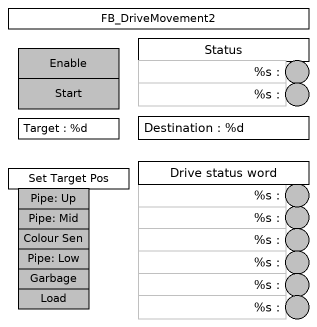
rectangle at (0,0)-(301,21): text "FB_DriveMovement2"
embedded screen at (130,30)-(301,311): FB_VC_Drive_Status
rectangle at (10,110)-(111,131): text "Target : %d"; shows $FB$.wTarget
rectangle at (10,40)-(111,71): text "Enable"; alarm colour if $FB$.bEnable; toggles $FB$.bEnable
rectangle at (10,70)-(111,101): text "Start"; alarm colour if $FB$.bStart; toggles $FB$.bStart
rectangle at (10,280)-(81,301): text "Load"; alarm colour if $FB$.wTarget = .GPOS_LOADING; runs INTERN ASSIGN $FB$.wTarget:=(GPOS_LOADING)
rectangle at (10,260)-(81,281): text "Garbage"; alarm colour if $FB$.wTarget = .GPOS_GARBAGE; runs INTERN ASSIGN $FB$.wTarget:=(GPOS_GARBAGE)
rectangle at (0,160)-(121,181): text "Set Target Pos"
rectangle at (10,240)-(81,261): text "Pipe: Low"; alarm colour if $FB$.wTarget = .GPOS_PIPE_LOW; runs INTERN ASSIGN $FB$.wTarget:=(GPOS_PIPE_LOW)
rectangle at (10,220)-(81,241): text "Colour Sen"; alarm colour if $FB$.wTarget = .GPOS_COLOR_SEN; runs INTERN ASSIGN $FB$.wTarget:=(GPOS_COLOR_SEN)
rectangle at (10,200)-(81,221): text "Pipe: Mid"; alarm colour if $FB$.wTarget = .GPOS_PIPE_MID; runs INTERN ASSIGN $FB$.wTarget:=(GPOS_PIPE_MID)
rectangle at (10,180)-(81,201): text "Pipe: Up"; alarm colour if $FB$.wTarget = .GPOS_PIPE_UP; runs INTERN ASSIGN $FB$.wTarget:=(GPOS_PIPE_UP)
1 more shapes without text or variables
*)

(* Visualisation FBs_Visu/FB_VC_Drive_Status
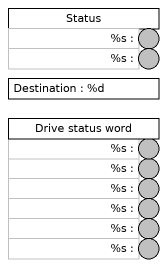
embedded screen at (0,150)-(151,171): VC_BOOLEANSTATUS
rectangle at (0,0)-(151,21): text "Status"
embedded screen at (0,170)-(151,191): VC_BOOLEANSTATUS
embedded screen at (0,130)-(151,151): VC_BOOLEANSTATUS
embedded screen at (0,190)-(151,211): VC_BOOLEANSTATUS
embedded screen at (0,210)-(151,231): VC_BOOLEANSTATUS
embedded screen at (0,230)-(151,251): VC_BOOLEANSTATUS
rectangle at (0,70)-(151,91): text "Destination : %d"; shows $FB$.wDestination
rectangle at (0,110)-(151,131): text "Drive status word"
embedded screen at (0,20)-(151,41): VC_BOOLEANSTATUS
embedded screen at (0,40)-(151,61): VC_BOOLEANSTATUS
*)

(* Visualisation Simulation/Simu_VC_Virtual_Ball
1 elements of other kinds (tables, trends, ...) not read
*)

(* Visualisation V_Drive
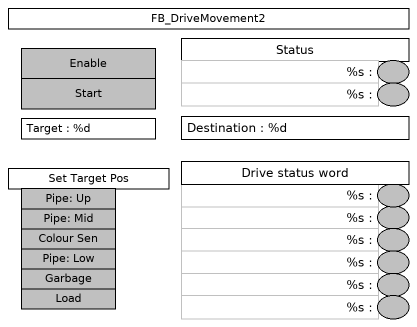
embedded screen at (0,0)-(401,311): FB_DriveMovement2
*)

(* Visualisation V_MAIN
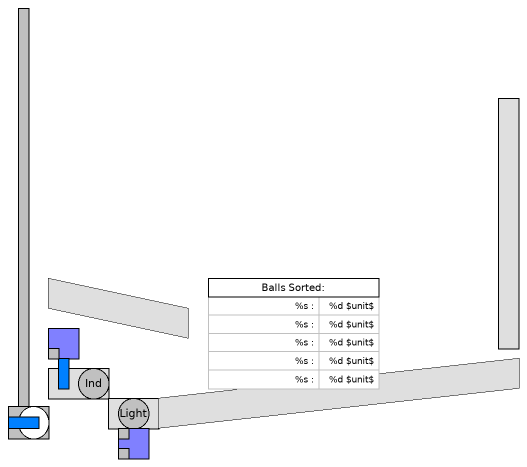
embedded screen at (60,320)-(531,451): VC_Graph_Sorter
embedded screen at (20,0)-(61,431): VC_Graph_Lift
embedded screen at (220,270)-(391,381): VC_Graph_Counters
2 more shapes without text or variables
*)

(* Visualisation V_VIRTUAL_MACHINE
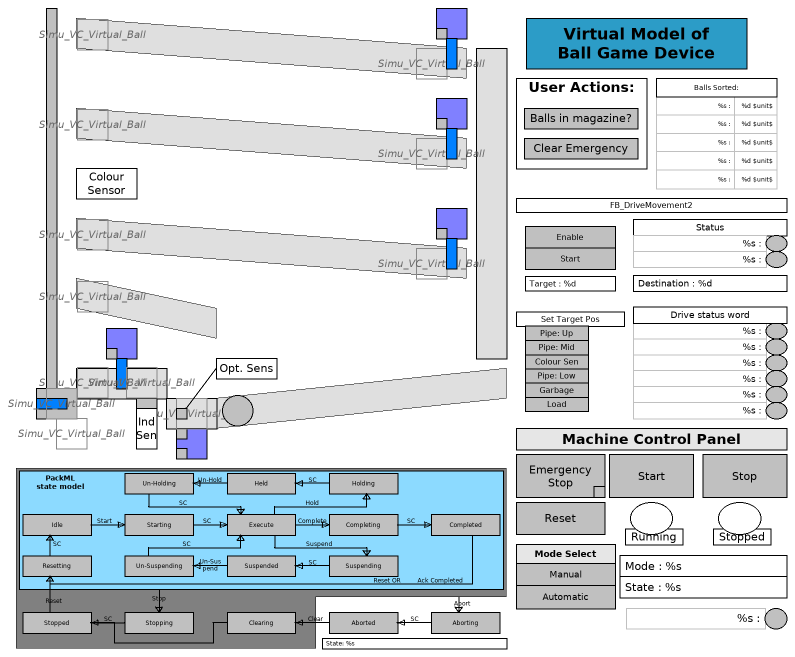
rectangle at (150,390)-(201,421): y offset -1 * PRG_HMI.iSorterLiftPos
rectangle at (100,350)-(111,381): invisible if .OSorterGate
rectangle at (120,390)-(141,401): alarm colour if .ISensorInd
rectangle at (160,420)-(171,431): alarm colour if .ISorterLiftUp
rectangle at (160,440)-(171,451): alarm colour if .ISorterLiftDown
rectangle at (90,340)-(101,351): alarm colour if .ISorterGateClosed
embedded screen at (160,390)-(191,421): Simu_VC_Virtual_Ball
rectangle at (160,400)-(171,411): alarm colour if .ISensorOpt
embedded screen at (110,359)-(141,390): Simu_VC_Virtual_Ball
embedded screen at (61,359)-(92,390): Simu_VC_Virtual_Ball
embedded screen at (40,410)-(71,441): Simu_VC_Virtual_Ball
rectangle at (20,380)-(61,411): y offset -1 * Simu_PRG_Simulation.iVirtualLiftPos
rectangle at (20,390)-(51,401): invisible if NOT .OEjector; y offset -1 * Simu_PRG_Simulation.iVirtualLiftPos
embedded screen at (30,380)-(61,411): Simu_VC_Virtual_Ball
embedded screen at (61,273)-(92,304): Simu_VC_Virtual_Ball
embedded screen at (61,211)-(92,242): Simu_VC_Virtual_Ball
embedded screen at (61,101)-(92,132): Simu_VC_Virtual_Ball
embedded screen at (61,11)-(92,42): Simu_VC_Virtual_Ball
embedded screen at (400,40)-(431,71): Simu_VC_Virtual_Ball
embedded screen at (400,130)-(431,161): Simu_VC_Virtual_Ball
embedded screen at (400,240)-(431,271): Simu_VC_Virtual_Ball
rectangle at (60,160)-(121,191): text "Colour / Sensor"
rectangle at (510,10)-(731,61): text "Virtual Model of / Ball Game Device"
rectangle at (120,400)-(141,441): text "Ind / Sen"
rectangle at (200,350)-(261,371): text "Opt. Sens"
ellipse at (206,387)-(237,418): invisible if NOT Simu_PRG_Simulation.bHasBallsInMagazine
embedded screen at (0,460)-(491,641): VC_PackMLStates
embedded screen at (640,70)-(761,181): VC_Graph_Counters
embedded screen at (500,190)-(771,411): FB_DriveMovement2
embedded screen at (500,420)-(771,601): VC_PANEL_MACHINECONTROL
rectangle at (420,220)-(431,231): alarm colour if .IGateClosedLow
rectangle at (420,110)-(431,121): alarm colour if .IGateClosedMid
rectangle at (420,20)-(431,31): alarm colour if .IGateClosedUp
rectangle at (430,120)-(441,151): invisible if .OGateMid
rectangle at (430,30)-(441,61): invisible if .OGateUp
rectangle at (430,230)-(441,261): invisible if .OGateLow
group at (500,70)-(631,161)
  rounded rectangle at (0,0)-(131,91): text "User Actions:"
  rounded rectangle at (8,30)-(122,51): text "Balls in magazine?"; alarm colour if Simu_PRG_Simulation.bHasBallsInMagazine; toggles Simu_PRG_Simulation.bHasBallsInMagazine
  rounded rectangle at (8,60)-(122,81): text "Clear Emergency"; alarm colour if NOT .IEmergencyClear; toggles .IEmergencyClear
embedded screen at (610,600)-(771,621): VC_BOOLEANSTATUS
19 more shapes without text or variables
*)

(* Visualisation Components/VC_BOOLEANSTATUS
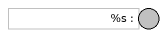
rectangle at (0,0)-(131,21): text "%s :"; shows $Name$
ellipse at (130,0)-(151,21): alarm colour if $bFlag$
*)

(* Visualisation Components/VC_Graph_Counters
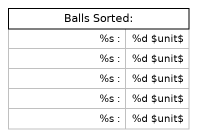
embedded screen at (0,20)-(181,41): VC_Var_Int
rectangle at (0,0)-(181,21): text "Balls Sorted:"
embedded screen at (0,40)-(181,61): VC_Var_Int
embedded screen at (0,60)-(181,81): VC_Var_Int
embedded screen at (0,80)-(181,101): VC_Var_Int
embedded screen at (0,100)-(181,121): VC_Var_Int
*)

(* Visualisation Components/VC_GRAPH_LIFT
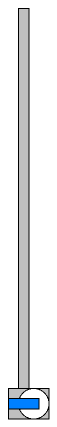
rectangle at (0,380)-(41,411): y offset -1 * PRG_HMI.iLiftPos
ellipse at (10,380)-(41,411): invisible if NOT .PRG_HMI.bBall_InLift; y offset -1 * PRG_HMI.iLiftPos
rectangle at (0,390)-(31,401): invisible if NOT .OEjector; y offset -1 * PRG_HMI.iLiftPos
1 more shapes without text or variables
*)

(* Visualisation Components/VC_GRAPH_SORTER
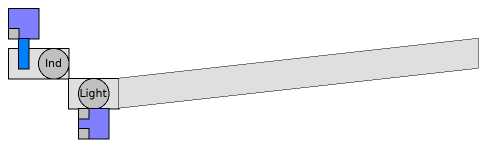
rectangle at (60,70)-(111,101): y offset -1 * PRG_HMI.iSorterLiftPos
rectangle at (10,30)-(21,61): invisible if .OSorterGate
ellipse at (70,70)-(101,101): text "Light"; alarm colour if .ISensorOpt; y offset -1 * PRG_HMI.iSorterLiftPos
ellipse at (30,40)-(61,71): text "Ind"; alarm colour if .ISensorInd
rectangle at (70,100)-(81,111): alarm colour if .ISorterLiftUp
rectangle at (70,120)-(81,131): alarm colour if .ISorterLiftDown
rectangle at (0,20)-(11,31): alarm colour if .ISorterGateClosed
6 more shapes without text or variables
*)

(* Visualisation Visual Components/VC_PackMLStates
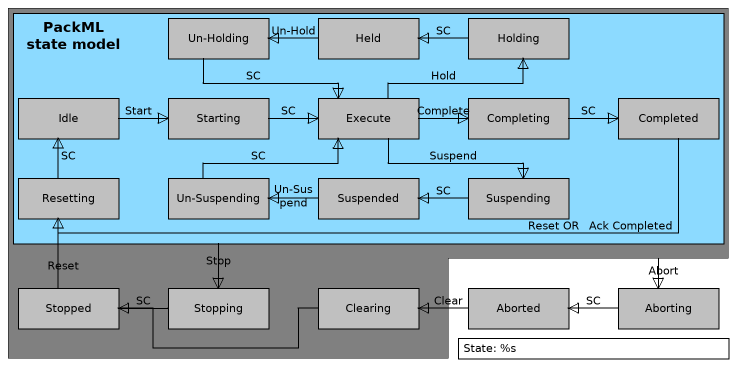
rounded rectangle at (160,280)-(261,321): text "Stopping"; alarm colour if $PackML$.eState = 4
rounded rectangle at (10,90)-(111,131): text "Idle"; alarm colour if $PackML$.eState = 6
rounded rectangle at (160,170)-(261,211): text "Un-Suspending"; alarm colour if $PackML$.eState = 11
rounded rectangle at (610,280)-(711,321): text "Aborting"; alarm colour if $PackML$.eState = 0
rounded rectangle at (460,280)-(561,321): text "Aborted"; alarm colour if $PackML$.eState = 1
rectangle at (450,330)-(721,351): text "State: %s"; shows .fbStateModel.eState
rounded rectangle at (310,280)-(411,321): text "Clearing"; alarm colour if $PackML$.eState = 2
rounded rectangle at (10,280)-(111,321): text "Stopped"; alarm colour if $PackML$.eState = 3
rounded rectangle at (10,170)-(111,211): text "Resetting"; alarm colour if $PackML$.eState = 5
rounded rectangle at (160,90)-(261,131): text "Starting"; alarm colour if $PackML$.eState = 7
rounded rectangle at (310,90)-(411,131): text "Execute"; alarm colour if $PackML$.eState = 8
rounded rectangle at (460,90)-(561,131): text "Completing"; alarm colour if $PackML$.eState = 15
rounded rectangle at (610,90)-(711,131): text "Completed"; alarm colour if $PackML$.eState = 16
rounded rectangle at (310,170)-(411,211): text "Suspended"; alarm colour if $PackML$.eState = 10
rounded rectangle at (460,170)-(561,211): text "Suspending"; alarm colour if $PackML$.eState = 9
rounded rectangle at (460,10)-(561,51): text "Holding"; alarm colour if $PackML$.eState = 12
rounded rectangle at (310,10)-(411,51): text "Held"; alarm colour if $PackML$.eState = 13
rounded rectangle at (160,10)-(261,51): text "Un-Holding"; alarm colour if $PackML$.eState = 14
polyline at (645,250)-(655,280): alarm colour if $PackML$.bAbort
rectangle at (635,255)-(676,271): text "Abort"; alarm colour if $PackML$.bAbort
polyline at (205,235)-(215,280): alarm colour if $PackML$.bStop
rectangle at (190,245)-(231,261): text "Stop"; alarm colour if $PackML$.bStop
polyline at (195,130)-(335,170): alarm colour if $PackML$.bSC
rectangle at (235,140)-(266,156): text "SC"; alarm colour if $PackML$.bSC
polyline at (195,50)-(335,90): alarm colour if $PackML$.bSC
polyline at (380,50)-(520,90): alarm colour if $PackML$.bHold
rectangle at (420,60)-(451,76): text "Hold"; alarm colour if $PackML$.bHold
polyline at (560,295)-(610,305): alarm colour if $PackML$.bSC
polyline at (45,210)-(55,280): alarm colour if $PackML$.bReset
polyline at (110,105)-(160,115): alarm colour if $PackML$.bStart
polyline at (110,295)-(310,340): alarm colour if $PackML$.bSC
rectangle at (230,60)-(261,76): text "SC"; alarm colour if $PackML$.bSC
polyline at (380,130)-(520,170): alarm colour if $PackML$.bSuspend
rectangle at (415,140)-(476,156): text "Suspend"; alarm colour if $PackML$.bSuspend
rectangle at (120,285)-(151,301): text "SC"; alarm colour if $PackML$.bSC
rectangle at (570,285)-(601,301): text "SC"; alarm colour if $PackML$.bSC
polyline at (410,295)-(460,305): alarm colour if $PackML$.bClear
rectangle at (420,285)-(461,301): text "Clear"; alarm colour if $PackML$.bClear
polyline at (260,105)-(310,115): alarm colour if $PackML$.bSC
rectangle at (265,95)-(296,111): text "SC"; alarm colour if $PackML$.bSC
rectangle at (110,95)-(151,111): text "Start"; alarm colour if $PackML$.bStart
rectangle at (35,250)-(76,266): text "Reset"; alarm colour if $PackML$.bReset
polyline at (410,185)-(460,195): alarm colour if $PackML$.bSC
rectangle at (420,175)-(451,191): text "SC"; alarm colour if $PackML$.bSC
polyline at (410,25)-(460,35): alarm colour if $PackML$.bSC
rectangle at (420,15)-(451,31): text "SC"; alarm colour if $PackML$.bSC
polyline at (260,185)-(310,195): alarm colour if $PackML$.bUn_Suspend
rectangle at (260,170)-(311,206): text "Un-Sus / pend"; alarm colour if $PackML$.bUn_Suspend
polyline at (260,25)-(310,35): alarm colour if $PackML$.bUn_Hold
rectangle at (260,15)-(311,31): text "Un-Hold"; alarm colour if $PackML$.bUn_Hold
polyline at (410,105)-(460,115): alarm colour if $PackML$.bComplete
rectangle at (410,95)-(461,111): text "Complete"; alarm colour if $PackML$.bComplete
polyline at (560,105)-(610,115): alarm colour if $PackML$.bSC
rectangle at (565,95)-(596,111): text "SC"; alarm colour if $PackML$.bSC
polyline at (45,130)-(55,170): alarm colour if $PackML$.bSC
rectangle at (45,140)-(76,156): text "SC"; alarm colour if $PackML$.bSC
polyline at (50,130)-(670,225): alarm colour if $PackML$.bReset OR $PackML$.Ack_Completed
rectangle at (515,210)-(576,226): text "Reset OR"; alarm colour if $PackML$.bReset
rectangle at (575,210)-(671,226): text "Ack Completed"; alarm colour if $PackML$.bAck_Completed
rectangle at (10,10)-(121,51): text "PackML / state model"
2 more shapes without text or variables
*)

(* Visualisation Simulator/MachineComponents/VC_PANEL_MACHINECONTROL
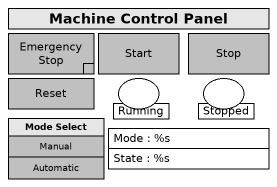
rounded rectangle at (0,25)-(86,66): text "Emergency / Stop"; alarm colour if .I_Btn_EStop; toggles .I_Btn_EStop
rounded rectangle at (90,25)-(171,66): text "Start"; alarm colour if .IRun; taps .I_Btn_Start
rounded rectangle at (0,70)-(86,101): text "Reset"; alarm colour if .I_Btn_Reset; taps .I_Btn_Reset
rectangle at (0,0)-(261,21): text "Machine Control Panel"
rectangle at (100,120)-(261,141): text "Mode : %s"; shows .fbStateModel.eMode
rectangle at (100,140)-(261,161): text "State : %s"; shows .fbStateModel.eState
embedded screen at (0,110)-(96,171): VC_Panel_ModeSelector
rectangle at (105,95)-(161,111): text "Running"
rectangle at (190,95)-(246,111): text "Stopped"
ellipse at (110,70)-(151,101): alarm colour if .O_Light_Start
ellipse at (195,70)-(236,101): alarm colour if .O_Light_Stop
embedded screen at (75,55)-(86,66): VC_sensor
rounded rectangle at (180,25)-(261,66): text "Stop"; alarm colour if .IRun; taps I_Btn_Stop
*)

(* Visualisation Simulator/MachineComponents/VC_PANEL_MODESELECTOR
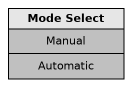
rounded rectangle at (0,20)-(116,46): text "Manual"; alarm colour if .HMI_uModeReq=3; runs INTERN ASSIGN HMI_uModeReq:=(3)
rectangle at (0,0)-(116,21): text "Mode Select"
rounded rectangle at (0,45)-(116,71): text "Automatic"; alarm colour if .HMI_uModeReq=1; runs INTERN ASSIGN HMI_uModeReq:=(1)
*)

(* Visualisation Components/VC_PIPE
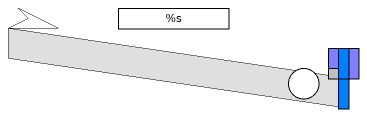
rectangle at (330,70)-(361,101): invisible if NOT .IPressureApplied
rectangle at (340,100)-(351,131): invisible if NOT $FB$.o_bGateIsClosed  OR NOT .IPressureApplied; toggles $FB$.i_bOpenGateCommand; tooltip Output cmd to open gate
rectangle at (330,90)-(341,101): alarm colour if $FB$.o_bGateIsClosed; tooltip Gate is closed input
polygon at (10,30)-(60,50): alarm colour if $FB$.i_bBallComingToPipe
ellipse at (290,90)-(321,121): alarm colour if $FB$.o_bBallExistInThePipe
rectangle at (120,30)-(231,51): text "%s"; shows $FB$.i_strPipeName
rectangle at (340,70)-(351,101): invisible if $FB$.o_bGateIsClosed; toggles $FB$.i_bOpenGateCommand; tooltip Output cmd to open gate
1 more shapes without text or variables
1 elements of other kinds (tables, trends, ...) not read
*)

(* Visualisation Simulator/Components/VC_sensor
rectangle at (0,0)-(11,11): alarm colour if $VAR$
*)

(* Visualisation Components/VC_Var_Int
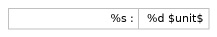
rectangle at (0,0)-(131,21): text "%s :"; shows $Name$
rectangle at (130,0)-(201,21): text "%d $unit$"; shows $VAR$
*)
